
FUNCTION CB_int_to_byte : BYTE

TITLE = ' Convert an integer into a byte '
VERSION : '1.0'
AUTHOR  : CB
NAME    : intToByt
FAMILY  : TNI

VAR_INPUT
    IN : INT;
END_VAR

BEGIN

CB_int_to_byte := INT_TO_BYTE(IN);

END_FUNCTION
